(*

.. <legal notes>

legal notes
=================
| SPDX-FileCopyrightText: © 2025 Oleksandr Tiutyk <trofimich@gmail.com>
| SPDX-License-Identifier: LGPL-3.0-only
| For details check: LGPL-3.0-only_

.. _LGPL-3.0-only: https://www.gnu.org/licenses/lgpl-3.0.en.html

.. </legal notes>

*)

{attribute 'no_explicit_call' := 'do not call this function block directly'} 
FUNCTION_BLOCK TaskSequence EXTENDS Task IMPLEMENTS ITaskSequence
VAR
	_ClassName : STRING := __POUNAME();

	_Tasks : TOF_Collections.List(0);
	
	_TaskSwitchingHandler : ITaskSwitchingHandler;
	
	_CurrentTaskIndex : DINT := -1;
END_VAR

METHOD AddTask : DINT
VAR_INPUT
	task : ITask;
END_VAR
VAR
	taskTypeNotSpecifiedException : TOF_Core.ArgumentNotSpecifiedException;
END_VAR
IF task = 0 THEN
	taskTypeNotSpecifiedException.Throw(Namespacename, ClassName, __POUNAME(), __POSITION(), 'task');
END_IF

_Tasks.AppendGeneric(GenericValueFactory.FromIObjectReference(task), index => AddTask);
END_METHOD

{attribute 'monitoring' := 'call'}
PROPERTY ClassName : STRING
GET
ClassName := _ClassName;
END_GET
END_PROPERTY

METHOD FINAL Clear
_Tasks.Clear();
END_METHOD

METHOD getTaskByIndex : ITask
VAR_INPUT
	taskIndex : DINT;
END_VAR
VAR
	taskInterface : TOF_Core.IObject;
	
	taskIndexOutOfRangeException : TOF_Core.ArgumentOutOfRangeException;
	
	toITaskConversionNotSupportedException : TOF_Core.StandardException;
END_VAR
IF taskIndex < 0 OR_ELSE taskIndex >= _Tasks.Count THEN
	taskIndexOutOfRangeException.Throw(NamespaceName, ClassName, __POUNAME(), __POSITION(), 'taskIndex', taskIndex);
END_IF

taskInterface := _Tasks.Get(taskIndex).AsIObject();

IF NOT __QUERYINTERFACE(taskInterface, getTaskByIndex) THEN
	toITaskConversionNotSupportedException.Throw(NamespaceName, ClassName, __POUNAME(), __POSITION(), "Can't convert task from _Tasks collection to ITask type");
END_IF
END_METHOD

{attribute 'monitoring' := 'call'}
PROPERTY NamespaceName : STRING
GET
NamespaceName := CurrentNamespace.Name;
END_GET
END_PROPERTY

METHOD PROTECTED OnCancel
VAR
	currentTask : ITask;
END_VAR
IF _CurrentTaskIndex > 0 AND_THEN _CurrentTaskIndex < _Tasks.Count THEN
	IF __QUERYINTERFACE(_Tasks.Get(_CurrentTaskIndex).AsIObject(), currentTask) THEN
		currentTask.Cancel();		
	END_IF
END_IF
END_METHOD

METHOD PROTECTED OnRunning 
VAR_INPUT
	startRequest : BOOL;
END_VAR
VAR_OUTPUT
	state : TASK_RUNNING_STATE;
	abortReason : WSTRING(255);
END_VAR
VAR
	currentTask, nextTask : ITask;
END_VAR
IF startRequest THEN	
	TOF_Core.LogManager.TryLogMessage("Task sequence starting", LOG_CATEGORY.INFORMATION, "TaskSequence", "TaskSequence.Starting");

	IF _Tasks.Count > 0 THEN
		_CurrentTaskIndex := 0;
		
		currentTask := getTaskByIndex(_CurrentTaskIndex);
		
		IF _TaskSwitchingHandler <> 0 THEN
			_TaskSwitchingHandler.OnNextTask(0, currentTask);
		END_IF
		
		currentTask.Start();
	ELSE
		state := TASK_RUNNING_STATE.DONE;
		RETURN;	
	END_IF
ELSE
	currentTask := getTaskByIndex(_CurrentTaskIndex);
	
	currentTask.Execute();	
END_IF

CHECK_TASK_COMPLETION:

IF currentTask.Aborted THEN
	state := TASK_RUNNING_STATE.ABORTED;
	abortReason := WideStringHelper.ConcatStrings255("Task '", currentTask.Name, "' aborted in queue");	

	TOF_Core.LogManager.TryLogMessage(abortReason, LOG_CATEGORY.INFORMATION, "TaskQueue", "TaskQueue.Task", "TaskQueue.Task.Aborted");	
ELSIF currentTask.Done THEN
	TOF_Core.LogManager.TryLogMessage(WideStringHelper.ConcatStrings255("Task '", currentTask.Name, "' done in sequence"), LOG_CATEGORY.INFORMATION, "TaskSequence", "TaskSequence.Task", "TaskSequence.Task.Done");

	IF _CurrentTaskIndex + 1 < _Tasks.Count THEN
		_CurrentTaskIndex := _CurrentTaskIndex + 1;
		
		nextTask := getTaskByIndex(_CurrentTaskIndex);
		
		IF _TaskSwitchingHandler <> 0 THEN			
			_TaskSwitchingHandler.OnNextTask(currentTask, nextTask);
		END_IF
		
		currentTask := nextTask;
		
		currentTask.Start();
		
		JMP CHECK_TASK_COMPLETION;
	ELSE
		IF _TaskSwitchingHandler <> 0 THEN			
			_TaskSwitchingHandler.OnNextTask(currentTask, 0);
		END_IF

		state := TASK_RUNNING_STATE.DONE;

		TOF_Core.LogManager.TryLogMessage("Task sequence done", LOG_CATEGORY.INFORMATION, "TaskSequence", "TaskSequence.Done");
	END_IF 
END_IF
END_METHOD

{attribute 'monitoring' := 'call'}
PROPERTY Size : ULINT
GET
Size := XSIZEOF(THIS^);
END_GET
END_PROPERTY

PROPERTY FINAL TaskCount : DINT
GET
TaskCount := _Tasks.Count;
END_GET
END_PROPERTY

PROPERTY FINAL TaskSwitchingHandler : ITaskSwitchingHandler
GET
TaskSwitchingHandler := _TaskSwitchingHandler;
END_GET
SET
_TaskSwitchingHandler := TaskSwitchingHandler;
END_SET
END_PROPERTY

END_FUNCTION_BLOCK

(* stored: Version 1.1.0.1
   POU TaskSequence: Id {57ebc80d-8e9e-4079-b23e-23120ddfa49e}, SpecialFunc None
   Folder Overriden members: Id {fa4015c4-9b09-4ca8-8a87-8fd2497e24b8}
   Folder Service members: Id {dfb1ef28-2e7d-45d9-a141-45600b7f6d77}
   Method AddTask: Id {4fbf566b-f914-4407-80d5-dd104cd557de}
   Property ClassName: Id {773ba440-b042-488f-97a2-de044245c5b8}
   Get Get: Id {c97bc7e4-1362-47f1-8cb5-39a5fff38a98}
   Method Clear: Id {d2f3a742-1eb6-4e3d-b5a5-c6bc001e8e97}
   Method getTaskByIndex: Id {db2a16e5-5db2-4e2b-93ea-bd2d371cec83}
   Property NamespaceName: Id {5dd6d568-afa1-4a66-a02b-252ca76934a5}
   Get Get: Id {b2f72abe-d7d0-40ef-aaed-f7660617931d}
   Method OnCancel: Id {7c8c6dde-1fe7-48db-9a57-8a23ac600474}
   Method OnRunning: Id {d440ee13-6872-4a06-96ce-9fcbf2169e4f}
   Property Size: Id {a6053151-483e-4238-9886-7e7b91664275}
   Get Get: Id {b11c9c5a-d14a-45ac-9b8c-29c4f081003a}
   Property TaskCount: Id {aadedd78-bdaf-4aac-af1e-c96cf8093b75}
   Get Get: Id {24847adc-b894-494f-b5f0-c26f6e5e9b2b}
   Property TaskSwitchingHandler: Id {9c42978d-d4f1-4caf-a41c-4ba59c2824fd}
   Get Get: Id {98b40666-63ec-4f03-9d44-478255ee8baf}
   Set Set: Id {d4b27105-8606-47f8-bdb2-54b0ddda9c46} *)
